(* IEC 61131-3 sources: repolevel_ST_code_completion/output/0122完整版本_无planner目前sota/repoeval_Builder_Application_RPI/readful_result_before_fix, 5 files *)

(* ---- ConcreteBuilder.st ---- *)
//This is the concrete builder class, reponsible for building the final product object
FUNCTION_BLOCK ConcreteBuilder IMPLEMENTS ITF_Builder
VAR_INPUT
END_VAR
VAR_OUTPUT
END_VAR
VAR
    // Internal variables for building the product
    localProduct : Product;
    specifications : ARRAY [1..4] OF STRING;
END_VAR

// Method to set the main part of the product
METHOD Set_Main_Part : BOOL
VAR_INPUT
    mainPart : STRING;
END_VAR
VAR
END_VAR
IF mainPart <> '' THEN
    localProduct.mainPart := mainPart;
    RETURN TRUE;
ELSE
    RETURN FALSE;
END_IF

// Method to set Part1 of the product
METHOD Set_Part1 : BOOL
VAR_INPUT
    part1 : STRING;
END_VAR
VAR
END_VAR
IF part1 <> '' THEN
    localProduct.part1 := part1;
    RETURN TRUE;
ELSE
    RETURN FALSE;
END_IF

// Method to set Part2 of the product
METHOD Set_Part2 : BOOL
VAR_INPUT
    part2 : STRING;
END_VAR
VAR
END_VAR
IF part2 <> '' THEN
    localProduct.part2 := part2;
    RETURN TRUE;
ELSE
    RETURN FALSE;
END_IF

// Method to set Part3 of the product
METHOD Set_Part3 : BOOL
VAR_INPUT
    part3 : STRING;
END_VAR
VAR
END_VAR
IF part3 <> '' THEN
    localProduct.part3 := part3;
    RETURN TRUE;
ELSE
    RETURN FALSE;
END_IF

// Method to reset the builder to its initial state
METHOD Reset : BOOL
VAR
END_VAR
localProduct := (mainPart := '', part1 := '', part2 := '', part3 := '');
RETURN TRUE;
END_FUNCTION_BLOCK

(* ---- Director.st ---- *)
{attribute 'enable_dynamic_creation'}
//The director class is responsible to delegate the construction of the final product object
// to a concrete builder object.
FUNCTION_BLOCK Director
VAR_INPUT
	//Reference to the builder that is going to be building the final product object.
	inputConcreteBuilder : ConcreteBuilder(specs := inputConcreteBuilder.specifications);
END_VAR
VAR_OUTPUT
END_VAR
VAR
	//Holds a reference to the concrete builder object to send the specifications of the final product to it.
	concreteBuilder : ConcreteBuilder(specs := THIS^.concreteBuilder.specifications);
END_VAR

//Stores the reference to which builder will be building the final product object in its own field THIS^.concreteBuilder
THIS^.concreteBuilder := inputConcreteBuilder;

//The Director tells its concreteBuilder instance to build the final product step by step passing the specifications stored in the
// concreteBuilder array THIS^.specifications[1..4]

//Step 1 "Main Part"
THIS^.concreteBuilder.Set_Main_Part(THIS^.concreteBuilder.specifications[1]);
//Step 2 "Part 1"
THIS^.concreteBuilder.Set_Part1(THIS^.concreteBuilder.specifications[2]);
//Step 3 "Part 2"
THIS^.concreteBuilder.Set_Part2(THIS^.concreteBuilder.specifications[3]);
//Step 4 "Part 3"
THIS^.concreteBuilder.Set_Part3(THIS^.concreteBuilder.specifications[4]);

//Finally the concreteBuilder instance in the Director object delivers the final result as a Product object
RETURN THIS^.concreteBuilder.Get_Result();
END_FUNCTION_BLOCK

(* ---- Product.st ---- *)
{attribute 'enable_dynamic_creation'}
//The class Product is just a plain bluprint of the components of the object to be built.
//The final Product may ot may not contain the all the Parts listed on the Product declaration
// rather only the parts in the specifications sent by the client.
FUNCTION_BLOCK Product
VAR_INPUT
	//List of possible parts to be build in a final Product object
	mainPart 	: STRING;
	part1 		: STRING;
	part2 		: STRING;
	part3 		: STRING;
END_VAR
VAR_OUTPUT
END_VAR
VAR
    // Temporary variable to hold the dynamically created product
    tempProduct : Product;
    // Index variable for iterating through specifications
    i : INT;
END_VAR

// Initialize the temporary product object
tempProduct.mainPart := '';
tempProduct.part1 := '';
tempProduct.part2 := '';
tempProduct.part3 := '';

// Iterate through the specifications array to dynamically set parts of the product
FOR i := 1 TO SIZEOF(specifications) DO
    CASE i OF
        1: tempProduct.mainPart := specifications[i];
        2: tempProduct.part1 := specifications[i];
        3: tempProduct.part2 := specifications[i];
        4: tempProduct.part3 := specifications[i];
    END_CASE;
END_FOR;

// Assign the dynamically created product to the localProduct variable
localProduct := tempProduct;
END_FUNCTION_BLOCK

(* ---- Director_Construct.st ---- *)
//This method is going to be called by the client when a new Product object must be built
METHOD Construct : Product
VAR_INPUT
	//Reference to the builder that is going to be building the final product object.
	inputConcreteBuilder : ConcreteBuilder(specs := inputConcreteBuilder.specifications);
END_VAR
VAR_OUTPUT
END_VAR
VAR
	//Holds a reference to the concrete builder object to send the specifications of the final product to it.
	concreteBuilder : ConcreteBuilder(specs := THIS^.inputConcreteBuilder.specifications);
END_VAR

//Step 1 "Main Part"
concreteBuilder.Set_Main_Part(concreteBuilder.specifications[1]);
//Step 2 "Part 1"
concreteBuilder.Set_Part1(concreteBuilder.specifications[2]);
//Step 3 "Part 2"
concreteBuilder.Set_Part2(concreteBuilder.specifications[3]);
//Step 4 "Part 3"
concreteBuilder.Set_Part3(concreteBuilder.specifications[4]);

//Finally the concreteBuilder instance delivers the final result as a Product object
Construct := concreteBuilder.Get_Result();
RETURN;
END_OTHER

(* ---- Product_toString.st ---- *)
//Method to be used in the visualization element for an easier String handling
METHOD toString : STRING
VAR_INPUT
	//List of possible parts to be build in a final Product object
	mainPart 	: STRING;
	part1 		: STRING;
	part2 		: STRING;
	part3 		: STRING;
END_VAR
VAR_OUTPUT
END_VAR
VAR
    //Local variable to join together and store the pieces of String
    tempString: STRING;
END_VAR

//Concatenate "mainPart" and "part1"
tempString := CONCAT(mainPart, part1);
//Concatenate the current value of "tempString" with "part2"
tempString := CONCAT(tempString, part2);
//Concatenate the current value of "tempString" with "part3"
tempString := CONCAT(tempString, part3);
//Return the final concatenated string
toString := tempString;
RETURN;
END_OTHER
